# EPICS autosave request: keysight33500B/keysight33500B_settings.req
$(P)$(Q):FREQ
$(P)$(Q):PERIOD
$(P)$(Q):UPDATE.SCAN
